// TIA Portal V15.1 export
// export: Created 2026-01-09T13:45:13.8678483Z, ExportSetting WithDefaults, WithReadOnly, DisplayName Totally Integrated Automation Portal, DisplayVersion V15.1 Update 8, DisplayName TIA Portal Openness, DisplayVersion V15.1 Update 8, DisplayName STEP 7 Professional, DisplayVersion V15.1 Update 8, DisplayName WinCC Advanced, DisplayVersion V15.1 Update 8
FUNCTION_BLOCK "6.WEIGHT_HANDLING"   // FB6, LAD
{ S7_Optimized_Access := 'TRUE' }
VERSION : 0.1
// stored: AutoNumber false, CodeModifiedDate 2025-08-27T17:12:27.5610885Z, CompileDate 2025-08-30T17:40:31.470686Z, CreationDate 2024-10-12T12:36:08.0193576Z, DownloadWithoutReinit false, HandleErrorsWithinBlock false, InterfaceModifiedDate 2023-12-29T17:39:18.5236469Z, IsConsistent true, IsIECCheckEnabled false, IsKnowHowProtected false, IsRetainMemResEnabled false, IsWriteProtected false, LibraryConformanceStatus The object is library-conformant., MemoryReserve 100, ModifiedDate 2025-08-27T17:12:27.5610885Z, ParameterModified 2023-11-29T03:49:57.2782849Z, PLCSimAdvancedSupport false, SetENOAutomatically False, StructureModified 2023-12-29T17:39:18.5236469Z, UDAEnableTagReadback false
   VAR_INPUT
      W_IN { ExternalAccessible := 'False'; ExternalVisible := 'False'; ExternalWritable := 'False'} : Real;
      WR_IN : Real;
      PV_IN1 : Real;
      PV_IN2 : Real;
      PV_IN3 : Real;
      PV_IN4 : Real;
      PV_IN5 : Real;
      PV_IN6 : Real;
      SV_IN1 : Real;
      SV_IN2 : Real;
      SV_IN3 : Real;
      SV_IN4 : Real;
      SV_IN5 : Real;
      SV_IN6 : Real;
      RUN_1 { ExternalAccessible := 'False'; ExternalVisible := 'False'; ExternalWritable := 'False'} : Bool;
      RUN_2 { ExternalAccessible := 'False'; ExternalVisible := 'False'; ExternalWritable := 'False'} : Bool;
      RUN_3 { ExternalAccessible := 'False'; ExternalVisible := 'False'; ExternalWritable := 'False'} : Bool;
      RUN_4 { ExternalAccessible := 'False'; ExternalVisible := 'False'; ExternalWritable := 'False'} : Bool;
      RUN_5 { ExternalAccessible := 'False'; ExternalVisible := 'False'; ExternalWritable := 'False'} : Bool;
      RUN_6 { ExternalAccessible := 'False'; ExternalVisible := 'False'; ExternalWritable := 'False'} : Bool;
      EMTY { ExternalAccessible := 'False'; ExternalVisible := 'False'; ExternalWritable := 'False'} : Bool;
   END_VAR
   VAR_OUTPUT
      W_OUT1 { ExternalAccessible := 'False'; ExternalVisible := 'False'; ExternalWritable := 'False'} : Real;
      W_OUT2 { ExternalAccessible := 'False'; ExternalVisible := 'False'; ExternalWritable := 'False'} : Real;
      W_OUT3 { ExternalAccessible := 'False'; ExternalVisible := 'False'; ExternalWritable := 'False'} : Real;
      W_OUT4 { ExternalAccessible := 'False'; ExternalVisible := 'False'; ExternalWritable := 'False'} : Real;
      W_OUT5 { ExternalAccessible := 'False'; ExternalVisible := 'False'; ExternalWritable := 'False'} : Real;
      W_OUT6 { ExternalAccessible := 'False'; ExternalVisible := 'False'; ExternalWritable := 'False'} : Real;
      "%W_OUT" { ExternalAccessible := 'False'; ExternalVisible := 'False'; ExternalWritable := 'False'} : Real;
   END_VAR
   VAR RETAIN
      W_Star : Real;
      W_Temp : Real;
   END_VAR
   VAR
      P_RUN1 : Bool;
      P_RUN2 : Bool;
      P_RUN3 : Bool;
      P_RUN4 : Bool;
      P_RUN5 : Bool;
      P_RUN6 : Bool;
      N_RUN1 : Bool;
      N_RUN2 : Bool;
      N_RUN3 : Bool;
      N_RUN4 : Bool;
      N_RUN5 : Bool;
      N_RUN6 : Bool;
   END_VAR
   VAR RETAIN
      PV1 : Real;
      PV2 : Real;
      PV3 : Real;
      PV4 : Real;
      PV5 : Real;
      PV6 : Real;
   END_VAR
   VAR_TEMP   // added for the SCL form of the ladder/FBD networks
      _w1 : Bool;
      _w2 : Bool;
      _w3 : Bool;
      _w4 : Bool;
      _w5 : Bool;
      _w6 : Bool;
   END_VAR
BEGIN

REGION Network 1
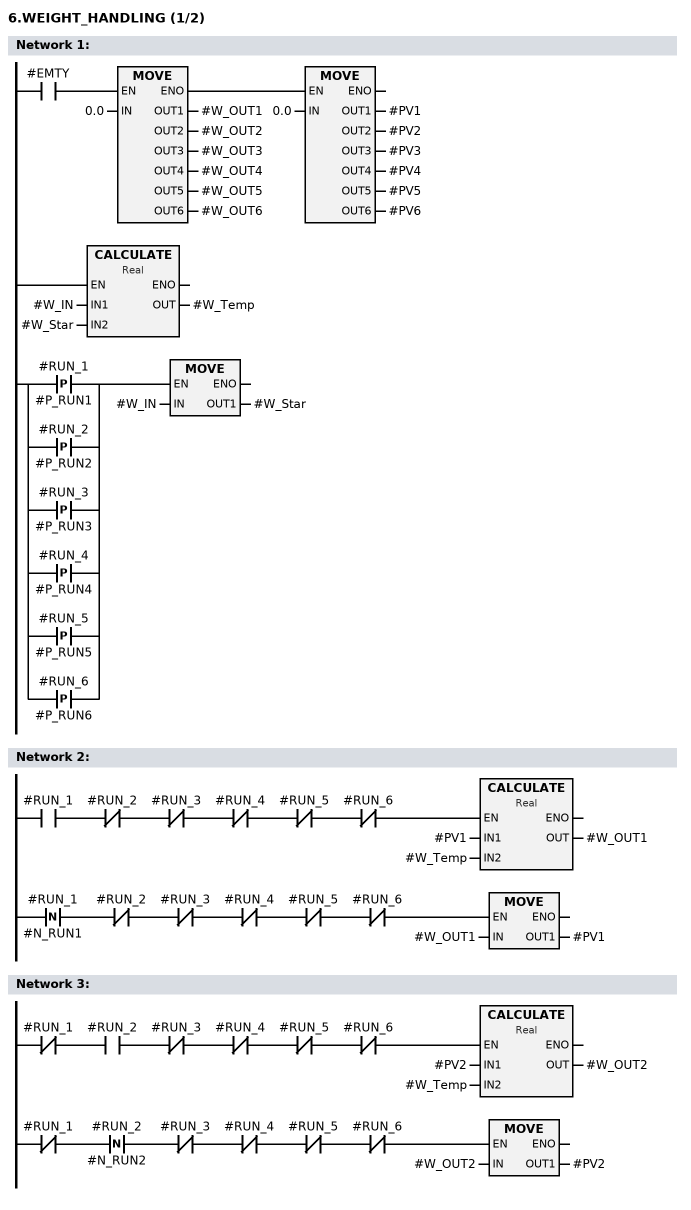
   RUNG wire#powerrail
      Contact( #EMTY )
      Move(in := 0.0, out1 => #W_OUT1, out2 => #W_OUT2, out3 => #W_OUT3, out4 => #W_OUT4, out5 => #W_OUT5, out6 => #W_OUT6)
      Move(in := 0.0, out1 => #PV1, out2 => #PV2, out3 => #PV3, out4 => #PV4, out5 => #PV5, out6 => #PV6)
   END_RUNG
   RUNG wire#powerrail
      { S7_Templates := "SrcType := Real"; S7_Expression := "IN1-IN2" } Calculate(in1 := #W_IN, in2 := #W_Star, out => #W_Temp)
   END_RUNG
   RUNG wire#powerrail
      P_Contact(operand := #RUN_1, bit := #P_RUN1)
      wire#w1
      Move(in := #W_IN, out1 => #W_Star)
   END_RUNG
   RUNG wire#powerrail
      P_Contact(operand := #RUN_2, bit := #P_RUN2)
   END_RUNG wire#w1
   RUNG wire#powerrail
      P_Contact(operand := #RUN_3, bit := #P_RUN3)
   END_RUNG wire#w1
   RUNG wire#powerrail
      P_Contact(operand := #RUN_4, bit := #P_RUN4)
   END_RUNG wire#w1
   RUNG wire#powerrail
      P_Contact(operand := #RUN_5, bit := #P_RUN5)
   END_RUNG wire#w1
   RUNG wire#powerrail
      P_Contact(operand := #RUN_6, bit := #P_RUN6)
   END_RUNG wire#w1
   // the same network as SCL:
   IF #EMTY THEN
       #W_OUT1 := 0.0;
       #W_OUT2 := 0.0;
       #W_OUT3 := 0.0;
       #W_OUT4 := 0.0;
       #W_OUT5 := 0.0;
       #W_OUT6 := 0.0;
       #PV1 := 0.0;
       #PV2 := 0.0;
       #PV3 := 0.0;
       #PV4 := 0.0;
       #PV5 := 0.0;
       #PV6 := 0.0;
   END_IF;
   #W_Temp := #W_IN-#W_Star;
   #_w1 := #RUN_1 AND NOT #P_RUN1;   // rising edge of #RUN_1
   #P_RUN1 := #RUN_1;
   #_w2 := #RUN_2 AND NOT #P_RUN2;   // rising edge of #RUN_2
   #P_RUN2 := #RUN_2;
   #_w3 := #RUN_3 AND NOT #P_RUN3;   // rising edge of #RUN_3
   #P_RUN3 := #RUN_3;
   #_w4 := #RUN_4 AND NOT #P_RUN4;   // rising edge of #RUN_4
   #P_RUN4 := #RUN_4;
   #_w5 := #RUN_5 AND NOT #P_RUN5;   // rising edge of #RUN_5
   #P_RUN5 := #RUN_5;
   #_w6 := #RUN_6 AND NOT #P_RUN6;   // rising edge of #RUN_6
   #P_RUN6 := #RUN_6;
   IF #_w1 OR #_w2 OR #_w3 OR #_w4 OR #_w5 OR #_w6 THEN #W_Star := #W_IN; END_IF;
END_REGION

REGION Network 2
   RUNG wire#powerrail
      Contact( #RUN_1 )
      I_Contact( #RUN_2 )
      I_Contact( #RUN_3 )
      I_Contact( #RUN_4 )
      I_Contact( #RUN_5 )
      I_Contact( #RUN_6 )
      { S7_Templates := "SrcType := Real"; S7_Expression := "IN1+IN2" } Calculate(in1 := #PV1, in2 := #W_Temp, out => #W_OUT1)
   END_RUNG
   RUNG wire#powerrail
      N_Contact(operand := #RUN_1, bit := #N_RUN1)
      I_Contact( #RUN_2 )
      I_Contact( #RUN_3 )
      I_Contact( #RUN_4 )
      I_Contact( #RUN_5 )
      I_Contact( #RUN_6 )
      Move(in := #W_OUT1, out1 => #PV1)
   END_RUNG
   // the same network as SCL:
   IF #RUN_1 AND NOT #RUN_2 AND NOT #RUN_3 AND NOT #RUN_4 AND NOT #RUN_5 AND NOT #RUN_6 THEN
       #W_OUT1 := #PV1+#W_Temp;
   END_IF;
   #_w1 := NOT #RUN_1 AND #N_RUN1;   // falling edge of #RUN_1
   #N_RUN1 := #RUN_1;
   IF #_w1 AND NOT #RUN_2 AND NOT #RUN_3 AND NOT #RUN_4 AND NOT #RUN_5 AND NOT #RUN_6 THEN
       #PV1 := #W_OUT1;
   END_IF;
END_REGION

REGION Network 3
   RUNG wire#powerrail
      I_Contact( #RUN_1 )
      Contact( #RUN_2 )
      I_Contact( #RUN_3 )
      I_Contact( #RUN_4 )
      I_Contact( #RUN_5 )
      I_Contact( #RUN_6 )
      { S7_Templates := "SrcType := Real"; S7_Expression := "IN1+IN2" } Calculate(in1 := #PV2, in2 := #W_Temp, out => #W_OUT2)
   END_RUNG
   RUNG wire#powerrail
      I_Contact( #RUN_1 )
      N_Contact(operand := #RUN_2, bit := #N_RUN2)
      I_Contact( #RUN_3 )
      I_Contact( #RUN_4 )
      I_Contact( #RUN_5 )
      I_Contact( #RUN_6 )
      Move(in := #W_OUT2, out1 => #PV2)
   END_RUNG
   // the same network as SCL:
   IF NOT #RUN_1 AND #RUN_2 AND NOT #RUN_3 AND NOT #RUN_4 AND NOT #RUN_5 AND NOT #RUN_6 THEN
       #W_OUT2 := #PV2+#W_Temp;
   END_IF;
   #_w1 := NOT #RUN_1 AND NOT #RUN_2 AND #N_RUN2;   // falling edge of #RUN_2
   #N_RUN2 := #RUN_2;
   IF #_w1 AND NOT #RUN_3 AND NOT #RUN_4 AND NOT #RUN_5 AND NOT #RUN_6 THEN #PV2 := #W_OUT2; END_IF;
END_REGION

REGION Network 4
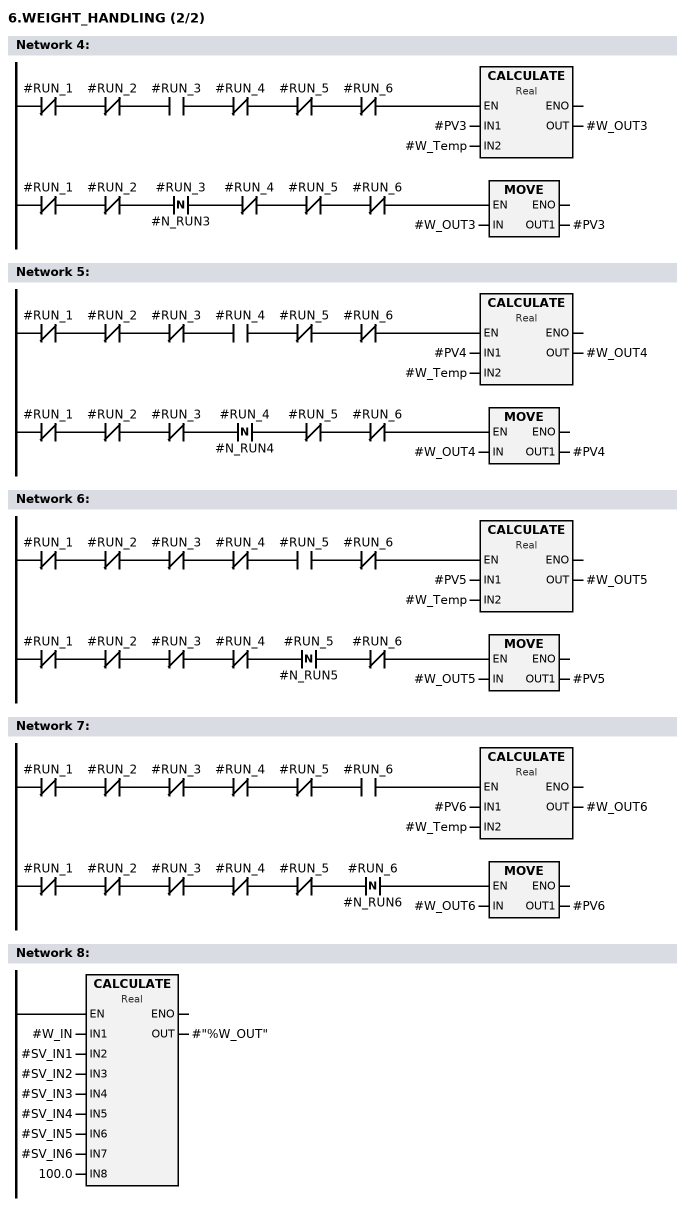
   RUNG wire#powerrail
      I_Contact( #RUN_1 )
      I_Contact( #RUN_2 )
      Contact( #RUN_3 )
      I_Contact( #RUN_4 )
      I_Contact( #RUN_5 )
      I_Contact( #RUN_6 )
      { S7_Templates := "SrcType := Real"; S7_Expression := "IN1+IN2" } Calculate(in1 := #PV3, in2 := #W_Temp, out => #W_OUT3)
   END_RUNG
   RUNG wire#powerrail
      I_Contact( #RUN_1 )
      I_Contact( #RUN_2 )
      N_Contact(operand := #RUN_3, bit := #N_RUN3)
      I_Contact( #RUN_4 )
      I_Contact( #RUN_5 )
      I_Contact( #RUN_6 )
      Move(in := #W_OUT3, out1 => #PV3)
   END_RUNG
   // the same network as SCL:
   IF NOT #RUN_1 AND NOT #RUN_2 AND #RUN_3 AND NOT #RUN_4 AND NOT #RUN_5 AND NOT #RUN_6 THEN
       #W_OUT3 := #PV3+#W_Temp;
   END_IF;
   #_w1 := NOT #RUN_1 AND NOT #RUN_2 AND NOT #RUN_3 AND #N_RUN3;   // falling edge of #RUN_3
   #N_RUN3 := #RUN_3;
   IF #_w1 AND NOT #RUN_4 AND NOT #RUN_5 AND NOT #RUN_6 THEN #PV3 := #W_OUT3; END_IF;
END_REGION

REGION Network 5
   RUNG wire#powerrail
      I_Contact( #RUN_1 )
      I_Contact( #RUN_2 )
      I_Contact( #RUN_3 )
      Contact( #RUN_4 )
      I_Contact( #RUN_5 )
      I_Contact( #RUN_6 )
      { S7_Templates := "SrcType := Real"; S7_Expression := "IN1+IN2" } Calculate(in1 := #PV4, in2 := #W_Temp, out => #W_OUT4)
   END_RUNG
   RUNG wire#powerrail
      I_Contact( #RUN_1 )
      I_Contact( #RUN_2 )
      I_Contact( #RUN_3 )
      N_Contact(operand := #RUN_4, bit := #N_RUN4)
      I_Contact( #RUN_5 )
      I_Contact( #RUN_6 )
      Move(in := #W_OUT4, out1 => #PV4)
   END_RUNG
   // the same network as SCL:
   IF NOT #RUN_1 AND NOT #RUN_2 AND NOT #RUN_3 AND #RUN_4 AND NOT #RUN_5 AND NOT #RUN_6 THEN
       #W_OUT4 := #PV4+#W_Temp;
   END_IF;
   #_w1 := NOT #RUN_1 AND NOT #RUN_2 AND NOT #RUN_3 AND NOT #RUN_4 AND #N_RUN4;   // falling edge of #RUN_4
   #N_RUN4 := #RUN_4;
   IF #_w1 AND NOT #RUN_5 AND NOT #RUN_6 THEN #PV4 := #W_OUT4; END_IF;
END_REGION

REGION Network 6
   RUNG wire#powerrail
      I_Contact( #RUN_1 )
      I_Contact( #RUN_2 )
      I_Contact( #RUN_3 )
      I_Contact( #RUN_4 )
      Contact( #RUN_5 )
      I_Contact( #RUN_6 )
      { S7_Templates := "SrcType := Real"; S7_Expression := "IN1+IN2" } Calculate(in1 := #PV5, in2 := #W_Temp, out => #W_OUT5)
   END_RUNG
   RUNG wire#powerrail
      I_Contact( #RUN_1 )
      I_Contact( #RUN_2 )
      I_Contact( #RUN_3 )
      I_Contact( #RUN_4 )
      N_Contact(operand := #RUN_5, bit := #N_RUN5)
      I_Contact( #RUN_6 )
      Move(in := #W_OUT5, out1 => #PV5)
   END_RUNG
   // the same network as SCL:
   IF NOT #RUN_1 AND NOT #RUN_2 AND NOT #RUN_3 AND NOT #RUN_4 AND #RUN_5 AND NOT #RUN_6 THEN
       #W_OUT5 := #PV5+#W_Temp;
   END_IF;
   #_w1 := NOT #RUN_1 AND NOT #RUN_2 AND NOT #RUN_3 AND NOT #RUN_4 AND NOT #RUN_5 AND #N_RUN5;   // falling edge of #RUN_5
   #N_RUN5 := #RUN_5;
   IF #_w1 AND NOT #RUN_6 THEN #PV5 := #W_OUT5; END_IF;
END_REGION

REGION Network 7
   RUNG wire#powerrail
      I_Contact( #RUN_1 )
      I_Contact( #RUN_2 )
      I_Contact( #RUN_3 )
      I_Contact( #RUN_4 )
      I_Contact( #RUN_5 )
      Contact( #RUN_6 )
      { S7_Templates := "SrcType := Real"; S7_Expression := "IN1+IN2" } Calculate(in1 := #PV6, in2 := #W_Temp, out => #W_OUT6)
   END_RUNG
   RUNG wire#powerrail
      I_Contact( #RUN_1 )
      I_Contact( #RUN_2 )
      I_Contact( #RUN_3 )
      I_Contact( #RUN_4 )
      I_Contact( #RUN_5 )
      N_Contact(operand := #RUN_6, bit := #N_RUN6)
      Move(in := #W_OUT6, out1 => #PV6)
   END_RUNG
   // the same network as SCL:
   IF NOT #RUN_1 AND NOT #RUN_2 AND NOT #RUN_3 AND NOT #RUN_4 AND NOT #RUN_5 AND #RUN_6 THEN
       #W_OUT6 := #PV6+#W_Temp;
   END_IF;
   #_w1 := NOT #RUN_1 AND NOT #RUN_2 AND NOT #RUN_3 AND NOT #RUN_4 AND NOT #RUN_5 AND NOT #RUN_6 AND #N_RUN6;   // falling edge of #RUN_6
   #N_RUN6 := #RUN_6;
   IF #_w1 THEN #PV6 := #W_OUT6; END_IF;
END_REGION

REGION Network 8
   RUNG wire#powerrail
      { S7_Templates := "SrcType := Real"; S7_Expression := "(IN1/(IN2+IN3+IN4+IN5+IN6+IN7))*IN8" } Calculate(in1 := #W_IN, in2 := #SV_IN1, in3 := #SV_IN2, in4 := #SV_IN3, in5 := #SV_IN4, in6 := #SV_IN5, in7 := #SV_IN6, in8 := 100.0, out => #"%W_OUT")
   END_RUNG
   // the same network as SCL:
   #"%W_OUT" := (#W_IN/(#SV_IN1+#SV_IN2+#SV_IN3+#SV_IN4+#SV_IN5+#SV_IN6))*100.0;
END_REGION
END_FUNCTION_BLOCK
